PROGRAM MAIN
VAR
END_VAR

PRG_TEST();

END_PROGRAM

(* stored: Version 1.1.0.1, ProductVersion 3.1.4024.11
   POU MAIN: Id {e26d26a9-6150-46eb-bf19-4ad3639df9c5}, SpecialFunc None *)
